FUNCTION_BLOCK SERVER_2_0 (* Connect to a CLIENT_0_2 Block *)
  (* Standard: 61499-2; Description: Copyright (c) 2017, 2025 fortiss GmbH , Johannes Kepler University Linz This program and the accompanying materials are made available under the terms of the Eclipse Public License 2.0 which is available at https://www.eclipse.org/legal/epl-2.0/ SPDX-License-Identifier: EPL-2.0 *)
  (* Version 3.0, 2025-09-26, Alois Zoitl, Created from SERVER_2 *)
  PACKAGE iec61499::net;
  {SET_ATTRIBUTE(eclipse4diac::core::GenericClassName, 'GEN_SERVER')}
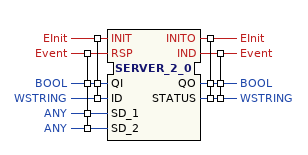
  EVENT_INPUT
    INIT : EInit WITH QI, ID; (* Enable Server for a Client connection (QI = TRUE) / Close Server (QI = FALSE) *)
    RSP WITH QI, SD_1, SD_2; (* Send data to Client *)
  END_EVENT
  EVENT_OUTPUT
    INITO : EInit WITH QO, STATUS; (* Ready for Client Connection (QI = TRUE) / Closed  (QI = FALSE) *)
    IND WITH QO, STATUS; (* New data available from Client *)
  END_EVENT
  VAR_INPUT
    QI : BOOL;
    ID : WSTRING;
    SD_1 : ANY;
    SD_2 : ANY;
  END_VAR
  VAR_OUTPUT
    QO : BOOL;
    STATUS : WSTRING;
  END_VAR
END_FUNCTION_BLOCK
